FUNCTION_BLOCK FB_NOTT_EVENTS
VAR_INPUT
END_VAR
VAR_OUTPUT
END_VAR
VAR
END_VAR

END_FUNCTION_BLOCK

(* stored: Version 1.1.0.1, ProductVersion 3.1.4024.14
   POU FB_NOTT_EVENTS: Id {bd6d6f12-a612-4c0f-ad91-f5fe8b2b3136}, SpecialFunc None *)
